FUNCTION_BLOCK FB_Template EXTENDS FD_Device IMPLEMENTS ITF_Convoyer
VAR_INPUT
END_VAR

VAR_OUTPUT
END_VAR

VAR
	
END_VAR


//******* Important and necessary
SUPER^();  
IF NOT Enable THEN RETURN; END_IF

//FB_Init ist immer implizit verfügbar und wird primär für die Initialisierung verwendet.
//Der Rückgabewert wird nicht ausgewertet. Für gezielte Einflussnahme können Sie
//die Methoden explizit deklarieren und darin mit dem Standard-Initialisierungscode 
//zusätzlichen Code bereitstellen. Sie können den Rückgabewert auswerten.
METHOD FB_Init: BOOL
VAR_INPUT    
	bInitRetains					: BOOL; 					// TRUE: Die Retain-Variablen werden initialisiert (Reset warm / Reset kalt)    
	bInCopyCode						: BOOL;  					// TRUE: Die Instanz wird danach in den Kopiercode kopiert (Online-Change)
	
	I_Name                : STRING;         //  Name
	I_ID                  : UINT;           // ID
  I_itfOwner					  : ITF_Owner;      // owner 
END_VAR
FB_ConvoyerDevice  FB_RouteDevice
END_METHOD

METHOD mAutomatic : E_CmdState
VAR_INPUT
	I_bExecute	: BOOL;
END_VAR
END_METHOD

METHOD mHold : E_CmdState
VAR_INPUT
	I_bExecute	: BOOL;
END_VAR
END_METHOD

METHOD mHome : E_CmdState
VAR_INPUT
	I_bExecute	: BOOL;
END_VAR
END_METHOD

METHOD mRelease : E_CmdState
VAR_INPUT
	I_bExecute	: BOOL;
END_VAR
END_METHOD

METHOD mSequence : E_CmdState
VAR_INPUT
	I_bExecute	: BOOL;
END_VAR
mSequence := SUPER^.mSequence(I_bExecute);	

//

CASE SequenceID OF

  //******************************************************* Idle 
  C_SeqStep_Idle: 
  	SequenceID       :=  C_SeqStep_Start;
  
  //****************************************************** Start
  C_SeqStep_Start:
   
  	SequenceID       :=  C_SeqStep_Done;
	
  C_SeqStep_Error: 
    //************* all FB reset

		//************* 
    mSequence := mDone(); 
  //**********************Done 
  	
 	C_SeqStep_Done:
  	mSequence := mDone();

END_CASE
END_METHOD

METHOD mService : E_CmdState
VAR_INPUT
	I_bExecute	: BOOL;
END_VAR
END_METHOD

METHOD mStop : E_CmdState
VAR_INPUT
	I_bExecute	: BOOL;
END_VAR
END_METHOD

END_FUNCTION_BLOCK

(* stored: Version 1.1.0.1, ProductVersion 3.1.4026.18
   POU FB_Template: Id {ce4fe2ee-cba5-47d7-b590-6780c2314c22}, SpecialFunc None
   Folder 01 Properties: Id {2c6c4302-16e3-4efb-964f-7d10c41dd0f2}
   Folder 02 Methodes: Id {d035e84b-6bed-4032-9638-02ba7e91191d}
   Method FB_Init: Id {382a709f-a145-4fc4-8162-73629f78573d}
   Method mAutomatic: Id {30d5cc96-2758-4ce6-b28f-ca28cae35736}
   Method mHold: Id {4f7534da-116a-4cb6-b0e2-caadc1e09ccf}
   Method mHome: Id {5bac2dfc-369d-493b-849c-3ddc789db988}
   Method mRelease: Id {b333511a-90e8-4d7a-bff1-01af1a22336e}
   Method mSequence: Id {80c4dc58-7709-4535-89bc-144e07f870b4}
   Method mService: Id {ac1a35cb-a794-423e-994f-b3a0921cf9ab}
   Method mStop: Id {0a1f33da-a07d-4338-8503-7cafc77bea19} *)
